TYPE ST_OpStates :
STRUCT
	Selected: BOOL;
	Ready: BOOL;
	Start: BOOL;
	Stop: BOOL;
	Reset: BOOL;
END_STRUCT
END_TYPE

(* stored: Version 1.1.0.1, ProductVersion 3.1.0.12
   DUT ST_OpStates: Id {ef675648-7f0e-4284-934d-70244ff185ed} *)
